FUNCTION_BLOCK FB_MAX_DT
  (* Standard: 61499-1 *)
  (* Version 0.1, 2006-09-12, JHC, Holobloc Inc, Moved to fb.rt.select. *)
  (* Version 0.0, 2004-12-15, JHC, Rockwell Automation, Converted from SRC format. *)
  (* Compiler header: package fb.rt.select; *)
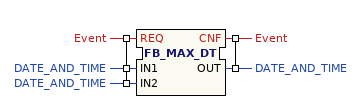
  EVENT_INPUT
    REQ WITH IN1, IN2;
  END_EVENT
  EVENT_OUTPUT
    CNF WITH OUT;
  END_EVENT
  VAR_INPUT
    IN1 : DATE_AND_TIME;
    IN2 : DATE_AND_TIME;
  END_VAR
  VAR_OUTPUT
    OUT : DATE_AND_TIME; (* MAX(IN1,IN2) *)
  END_VAR
END_FUNCTION_BLOCK
